// TIA Portal V15.1 export
// export: Created 2024-06-21T08:40:53.306712Z, ExportSetting WithDefaults, DisplayName Totally Integrated Automation Portal, DisplayVersion V15.1 Update 5, DisplayName TIA Portal Openness, DisplayVersion V15.1 Update 5, DisplayName SINAMICS Startdrive Advanced, DisplayVersion V15.1, DisplayName G130, G150, S120, S150, SINAMICS MV, S210, DisplayVersion V15.1, DisplayName G110M, G120, G120C, G120D, G120P, DisplayVersion V15.1, DisplayName STEP 7 Professional, DisplayVersion V15.1 Update 5, DisplayName STEP 7 Safety, DisplayVersion V15.1, DisplayName WinCC Professional, DisplayVersion V15.1 Update 5, DisplayName SIMATIC Visualization Architect, DisplayVersion V15.1
FUNCTION_BLOCK "LPulsesGenerator"   // FB1010, FBD
TITLE = LPulsesGenerator
{ S7_Optimized_Access := 'FALSE' }
AUTHOR : VCC
FAMILY : Control
NAME : PulseGen
VERSION : 1.0
// ================================================================================
// LPulsesGenerator is used everywhere a pulse signal is requiered.
// This function is able to generate pulse without disturbance due to scan time of 
// CPU. This function is able to generate pulse with a fix frequency.
// This function is also able to generate pulse with a defined time ON and a 
// different Time OFF.
// It is also possible to hold the function.
// It is also possible to use the running value of time ON and time OFF.
// ================================================================================
// stored: AutoNumber false, IsIECCheckEnabled false, SetENOAutomatically False, UDAEnableTagReadback false
   VAR_INPUT
      I_Input { ExternalAccessible := 'False'; ExternalVisible := 'False'; ExternalWritable := 'False'} : Bool;   // Input to start pulse generator
      I_Hold { ExternalAccessible := 'False'; ExternalVisible := 'False'; ExternalWritable := 'False'} : Bool;   // Input to hold the pulse generator
      I_Frequency { ExternalAccessible := 'False'; ExternalVisible := 'False'; ExternalWritable := 'False'} : DInt;   // Input to generated pulses to this frequency
      I_TimeOFF { ExternalAccessible := 'False'; ExternalVisible := 'False'; ExternalWritable := 'False'} : DInt;   // Duration OFF for pulses
      I_TimeON { ExternalAccessible := 'False'; ExternalVisible := 'False'; ExternalWritable := 'False'} : DInt;   // Duration ON for pulses
   END_VAR
   VAR_OUTPUT
      O_Pulses { ExternalAccessible := 'False'; ExternalVisible := 'False'; ExternalWritable := 'False'} : Bool;   // Pulses
      O_TimeOFF { ExternalAccessible := 'False'; ExternalVisible := 'False'; ExternalWritable := 'False'} : DInt;   // Value TimerOFF period
      O_TimeON { ExternalAccessible := 'False'; ExternalVisible := 'False'; ExternalWritable := 'False'} : DInt;   // Value TimerON period
   END_VAR
   VAR DB_SPECIFIC
      OFF_Finished { ExternalAccessible := 'False'; ExternalVisible := 'False'; ExternalWritable := 'False'} : Bool;   // Signal when timer OFF period finished
      ON_Finished { ExternalAccessible := 'False'; ExternalVisible := 'False'; ExternalWritable := 'False'} : Bool;   // Signal when timer ON period finished
      TimeOFF { ExternalAccessible := 'False'; ExternalVisible := 'False'; ExternalWritable := 'False'} : DInt;   // Duration OFF for pulses
      TimeON { ExternalAccessible := 'False'; ExternalVisible := 'False'; ExternalWritable := 'False'} : DInt;   // Duration ON for pulses
      OFF_FinishPulse { ExternalAccessible := 'False'; ExternalVisible := 'False'; ExternalWritable := 'False'} : Bool;   // Off Finished pulse
      RunningTimeOFF { ExternalAccessible := 'False'; ExternalVisible := 'False'; ExternalWritable := 'False'} : DInt;   // Duration OFF for pulses
      TimeOffOT { ExternalAccessible := 'False'; ExternalVisible := 'False'; ExternalWritable := 'False'} : DInt;   // Overtime for timer off
      TimeOffOTAcc { ExternalAccessible := 'False'; ExternalVisible := 'False'; ExternalWritable := 'False'} : DInt;   // Acculumated overtime for timer off
      TimeOffAdj { ExternalAccessible := 'False'; ExternalVisible := 'False'; ExternalWritable := 'False'} : DInt;   // Adjusted value for Timer off
      ON_FinishPulse { ExternalAccessible := 'False'; ExternalVisible := 'False'; ExternalWritable := 'False'} : Bool;   // On Finished pulse
      RunningTimeON { ExternalAccessible := 'False'; ExternalVisible := 'False'; ExternalWritable := 'False'} : DInt;   // Duration OFF for pulses
      TimeOnOT { ExternalAccessible := 'False'; ExternalVisible := 'False'; ExternalWritable := 'False'} : DInt;   // Overtime for timer on
      TimeOnOTAcc { ExternalAccessible := 'False'; ExternalVisible := 'False'; ExternalWritable := 'False'} : DInt;   // Acculumated overtime for timer on
      TimeOnAdj { ExternalAccessible := 'False'; ExternalVisible := 'False'; ExternalWritable := 'False'} : DInt;   // Adjusted value for Timer on
   END_VAR
   VAR
      TimerOFFPer { ExternalAccessible := 'False'; ExternalVisible := 'False'; ExternalWritable := 'False'; S7_SetPoint := 'True'} : "LTimer";   // Timer OFF period
      TimerONPer { ExternalAccessible := 'False'; ExternalVisible := 'False'; ExternalWritable := 'False'; S7_SetPoint := 'True'} : "LTimer";   // Timer ON period
   END_VAR
   VAR_TEMP
      Frequency : DInt;   // Temp frequency
   END_VAR
   VAR_TEMP   // added for the SCL form of the ladder/FBD networks
      _w1 : Bool;
      _w2 : Bool;
   END_VAR
BEGIN

REGION Network 1: **** 4.4 - Machine Status - Calculated **** Reset all timer values
   // Reset all timer values
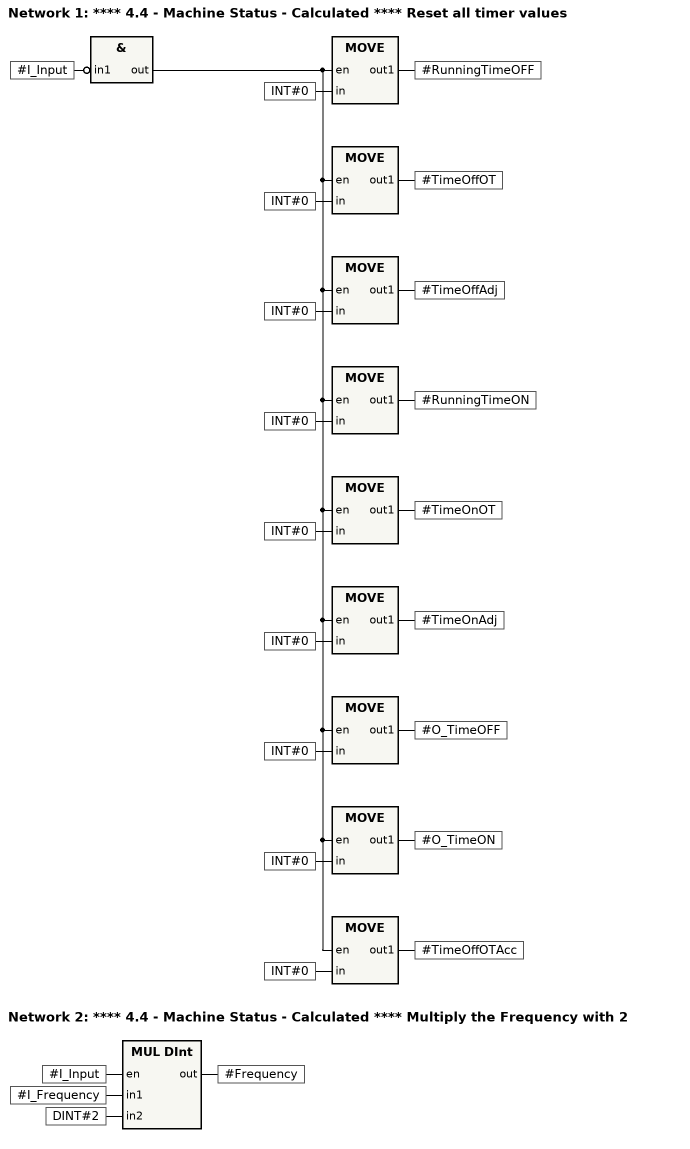
   IF NOT #I_Input THEN
       #RunningTimeOFF := INT#0;
       #TimeOffOT := INT#0;
       #TimeOffAdj := INT#0;
       #RunningTimeON := INT#0;
       #TimeOnOT := INT#0;
       #TimeOnAdj := INT#0;
       #O_TimeOFF := INT#0;
       #O_TimeON := INT#0;
       #TimeOffOTAcc := INT#0;
   END_IF;
END_REGION

REGION Network 2: **** 4.4 - Machine Status - Calculated **** Multiply the Frequency with 2
   // Multiply the Frequency with 2
   IF #I_Input THEN #Frequency := #I_Frequency * DINT#2; END_IF;
END_REGION

REGION Network 3: **** 4.4 - Machine Status - Calculated **** Calculation of TimeOFF and TimeON if I_Frequemcy selected
   // Calculation of TimeOFF and TimeON if I_Frequemcy selected
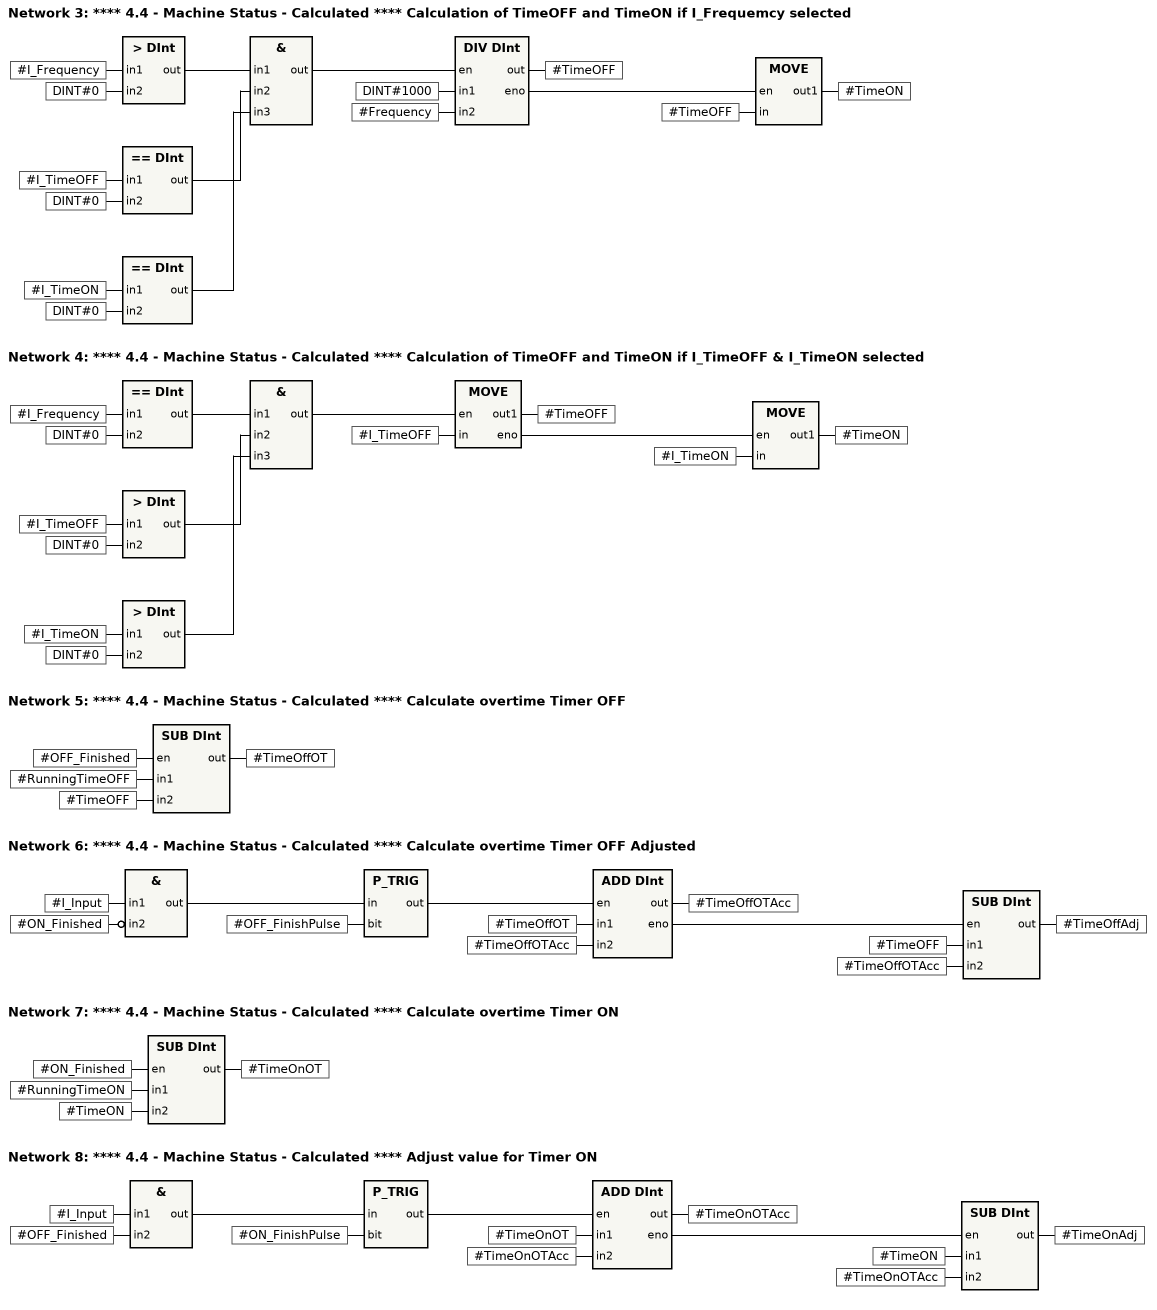
   // ENO of a box is taken as its EN; it also drops when the box reports an error
   IF (#I_Frequency > DINT#0) AND (#I_TimeOFF = DINT#0) AND (#I_TimeON = DINT#0) THEN
       #TimeOFF := DINT#1000 / #Frequency;
       #TimeON := #TimeOFF;
   END_IF;
END_REGION

REGION Network 4: **** 4.4 - Machine Status - Calculated **** Calculation of TimeOFF and TimeON if I_TimeOFF & I_TimeON selected
   // Calculation of TimeOFF and TimeON if I_TimeOFF & I_TimeON selected
   // ENO of a box is taken as its EN; it also drops when the box reports an error
   IF (#I_Frequency = DINT#0) AND (#I_TimeOFF > DINT#0) AND (#I_TimeON > DINT#0) THEN
       #TimeOFF := #I_TimeOFF;
       #TimeON := #I_TimeON;
   END_IF;
END_REGION

REGION Network 5: **** 4.4 - Machine Status - Calculated **** Calculate overtime Timer OFF
   // Calculate overtime Timer OFF
   IF #OFF_Finished THEN #TimeOffOT := #RunningTimeOFF - #TimeOFF; END_IF;
END_REGION

REGION Network 6: **** 4.4 - Machine Status - Calculated **** Calculate overtime Timer OFF Adjusted
   // Calculate overtime Timer OFF Adjusted
   // ENO of a box is taken as its EN; it also drops when the box reports an error
   #_w1 := #I_Input AND NOT #ON_Finished;
   #_w2 := #_w1 AND NOT #OFF_FinishPulse;   // rising edge
   #OFF_FinishPulse := #_w1;
   IF #_w2 THEN
       #TimeOffOTAcc := #TimeOffOT + #TimeOffOTAcc;
       #TimeOffAdj := #TimeOFF - #TimeOffOTAcc;
   END_IF;
END_REGION

REGION Network 7: **** 4.4 - Machine Status - Calculated **** Calculate overtime Timer ON
   // Calculate overtime Timer ON
   IF #ON_Finished THEN #TimeOnOT := #RunningTimeON - #TimeON; END_IF;
END_REGION

REGION Network 8: **** 4.4 - Machine Status - Calculated **** Adjust value for Timer ON
   // Adjust value for Timer ON
   // ENO of a box is taken as its EN; it also drops when the box reports an error
   #_w1 := #I_Input AND #OFF_Finished;
   #_w2 := #_w1 AND NOT #ON_FinishPulse;   // rising edge
   #ON_FinishPulse := #_w1;
   IF #_w2 THEN
       #TimeOnOTAcc := #TimeOnOT + #TimeOnOTAcc;
       #TimeOnAdj := #TimeON - #TimeOnOTAcc;
   END_IF;
END_REGION

REGION Network 9: **** 4.4 - Machine Status - Calculated **** Timer to generated Time OFF
   // Timer to generated Time OFF
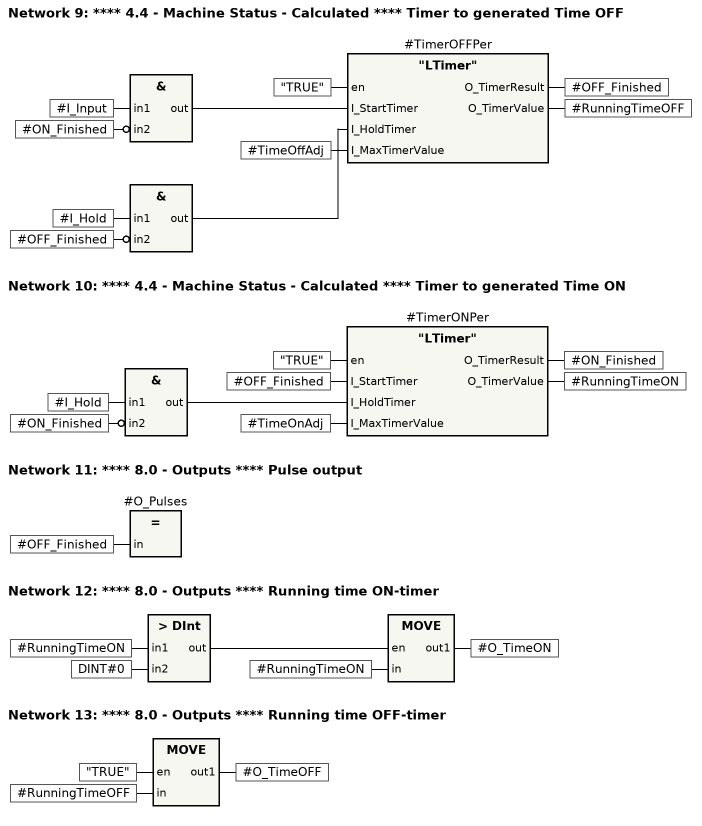
   IF "TRUE" THEN
       #TimerOFFPer(I_StartTimer := #I_Input AND NOT #ON_Finished,   // "LTimer"
                    I_HoldTimer := #I_Hold AND NOT #OFF_Finished,
                    I_MaxTimerValue := #TimeOffAdj,
                    O_TimerResult => #OFF_Finished,
                    O_TimerValue => #RunningTimeOFF);
   END_IF;
END_REGION

REGION Network 10: **** 4.4 - Machine Status - Calculated **** Timer to generated Time ON
   // Timer to generated Time ON
   IF "TRUE" THEN
       #TimerONPer(I_StartTimer := #OFF_Finished,   // "LTimer"
                   I_HoldTimer := #I_Hold AND NOT #ON_Finished,
                   I_MaxTimerValue := #TimeOnAdj,
                   O_TimerResult => #ON_Finished,
                   O_TimerValue => #RunningTimeON);
   END_IF;
END_REGION

REGION Network 11: **** 8.0 - Outputs **** Pulse output
   // Pulse output
   #O_Pulses := #OFF_Finished;
END_REGION

REGION Network 12: **** 8.0 - Outputs **** Running time ON-timer
   // Running time ON-timer
   IF #RunningTimeON > DINT#0 THEN #O_TimeON := #RunningTimeON; END_IF;
END_REGION

REGION Network 13: **** 8.0 - Outputs **** Running time OFF-timer
   // Running time OFF-timer
   IF "TRUE" THEN #O_TimeOFF := #RunningTimeOFF; END_IF;
END_REGION
END_FUNCTION_BLOCK
